TYPE ST_BaseHMITopElement_Command :
STRUCT
END_STRUCT
END_TYPE

(* stored: Version 1.1.0.1
   DUT ST_BaseHMITopElement_Command: Id {12071bf1-15b1-0080-2afe-79715ca4bddf} *)
